INTERFACE ITestEventHandler EXTENDS IEventHandlerBase

METHOD OnCustomEvent
VAR_INPUT
    EventData : UDINT;
END_VAR
END_METHOD

END_INTERFACE

(* stored: Version 1.1.0.1, ProductVersion 3.1.4024.3
   Itf ITestEventHandler: Id {9ee385fc-e8f7-4d68-bb53-356119ae705f}
   Method OnCustomEvent: Id {421a15e4-156d-4b3c-bbf9-040d84929891} *)
